FUNCTION_BLOCK FB_ORG_PositiveEndLessByTouchprobe
VAR_INPUT
	Axis		:AXIS_REF;
	Execute		:BOOL;
	Position	:LREAL;
	Velocity	:LREAL;
END_VAR
VAR_OUTPUT
	Error	:BOOL;
	Busy	:BOOL;
	Done	:BOOL;
END_VAR
VAR
	nStep	:INT;
	fbTrig	:R_TRIG;
	fbMC_MoveVelocity: MC_MoveVelocity;
	MC_TouchProbe: MC_TouchProbe;
	MC_AbortTrigger: MC_AbortTrigger;
	TRIGGER_REF	:TRIGGER_REF ;
	MC_ReadDriveAddress: MC_ReadDriveAddress;
	MC_Stop: MC_Stop;
	MC_Home: MC_Home;
	MC_SetPosition: MC_SetPosition;
END_VAR

fbTrig(CLK:=Execute);
Axis.ReadStatus();

IF fbTrig.Q THEN

	IF Axis.Status.StandStill THEN
		MC_ReadDriveAddress(Axis:= Axis,Execute:=FALSE);
		nStep	:=1;
	ELSE
		nStep	:= 99;
	END_IF;	
END_IF
		
CASE nStep OF
	1:		
		Busy:= TRUE;
		MC_ReadDriveAddress(
			Axis:= Axis, 
			Execute:=TRUE , 
			Done=> , 
			Busy=> , 
			Error=> , 
			ErrorID=> , 
			DriveAddress=> );
	IF MC_ReadDriveAddress.Done THEN
		Intial();
		nStep	:= 5;
	END_IF
5:
			MC_TouchProbe(
				Axis:= Axis, 
				TriggerInput:=TRIGGER_REF , 
				Execute:= TRUE, 
				WindowOnly:= , 
				FirstPosition:= , 
				LastPosition:= , 
				Done=> , 
				Busy=> , 
				CommandAborted=> , 
				Error=> , 
				ErrorID=> , 
				RecordedPosition=> , 
				RecordedData=> );	
			fbMC_MoveVelocity(
				Axis:= Axis, 
				Execute:= MC_TouchProbe.Busy, 
				Velocity:= Velocity, 
				Acceleration:= , 
				Deceleration:= , 
				Jerk:= , 
				Direction:= , 
				BufferMode:= , 
				Options:= , 
				InVelocity=> , 
				Busy=> , 
				Active=> , 
				CommandAborted=> , 
				Error=> , 
				ErrorID=> );	
		
			MC_Stop(
				Axis:= Axis, 
				Execute:=MC_TouchProbe.Done , 
				Deceleration:= , 
				Jerk:= , 
				Options:= , 
				Done=> , 
				Busy=> , 
				Active=> , 
				CommandAborted=> , 
				Error=> , 
				ErrorID=> );
			IF Axis.Status.MotionState = MC_AXISSTATE_STOPPING THEN	
				nStep	:= 10;
				END_IF;
10:	
	IF Axis.Status.MotionState = MC_AXISSTATE_STANDSTILL THEN
		nStep	:= 15;
	END_IF
			MC_Stop(
				Axis:= Axis, 
				Execute:= FALSE, 
				Deceleration:= , 
				Jerk:= , 
				Options:= , 
				Done=> , 
				Busy=> , 
				Active=> , 
				CommandAborted=> , 
				Error=> , 
				ErrorID=> );
	15:
		MC_SetPosition(
		Axis:= Axis, 
		Execute:= TRUE, 
		Position:=Axis.NcToPlc.ActPos - MC_TouchProbe.RecordedPosition ,
		Mode:= , 
		Options:= , 
		Done=> , 
		Busy=> , 
		Error=> , 
		ErrorID=> );
	IF MC_SetPosition.Done	THEN
		MC_Home.Execute:=TRUE;
	END_IF
	MC_Home(
		Axis:= Axis, 
		Execute:= , 
		Position:=(Axis.NcToPlc.ActPos - MC_TouchProbe.RecordedPosition) - Position, 
		HomingMode:= MC_ForceCalibration, 
		BufferMode:= , 
		Options:= , 
		bCalibrationCam:= , 
		Done=> , 
		Busy=> , 
		Active=> , 
		CommandAborted=> , 
		Error=> , 
		ErrorID=> );
	IF MC_Home.Done	THEN
		nStep:=20;
	END_IF
	20:
	Busy	:=FALSE;
	Done	:=TRUE;		
	IF NOT Execute THEN
		Done	:=FALSE;		
		nStep	:= 0;
	END_IF
END_CASE

METHOD FB_init : BOOL
VAR_INPUT
	bInitRetains : BOOL; // if TRUE, the retain variables are initialized (warm start / cold start)
	bInCopyCode : BOOL;  // if TRUE, the instance afterwards gets moved into the copy code (online change)
END_VAR
END_METHOD

METHOD INTERNAL Intial : BOOL
VAR_INPUT
END_VAR
TRIGGER_REF.EncoderID			:= Axis.DriveAddress.NcAxisId;
TRIGGER_REF.TouchProbe			:= Tc2_MC2.TouchProbe1;
TRIGGER_REF.SignalSource		:= Tc2_MC2.SignalSource_Default;
TRIGGER_REF.Mode				:= Tc2_MC2.TOUCHPROBEMODE_SINGLE;

	fbMC_MoveVelocity(Axis:= Axis, Execute:= FALSE);
	MC_TouchProbe(Axis:= Axis,TriggerInput:=TRIGGER_REF ,Execute:= FALSE);
	MC_AbortTrigger(Axis:= Axis,TriggerInput:=TRIGGER_REF ,Execute:= FALSE);
	MC_ReadDriveAddress(Axis:= Axis, Execute:= FALSE);
	MC_Stop(Axis:= Axis, Execute:= FALSE);
	MC_Home(Axis:= Axis, Execute:= FALSE);
	MC_SetPosition(Axis:= Axis, Execute:= FALSE);
END_METHOD

END_FUNCTION_BLOCK

(* stored: Version 1.1.0.1, ProductVersion 3.1.4024.15
   POU FB_ORG_PositiveEndLessByTouchprobe: Id {faa075a7-dd9a-48eb-8cfa-3ac468207e94}, SpecialFunc None
   Method FB_init: Id {fc414f99-1aaf-4274-8ed2-37a06a6b9003}
   Method Intial: Id {bb6f6f65-7289-449f-a1bc-8df3f95e5749} *)
